ORGANIZATION_BLOCK OB 1
BEGIN
	CALL	FC 1
END_ORGANIZATION_BLOCK

FUNCTION FC 1 : VOID
BEGIN
	CALL	FC 1
END_FUNCTION
